Staubli VAL3: Wizard_bigBox.pgx

program Wizard_bigBox()
begin
end
